Universal Robots PolyScope program: nastrobello.urp

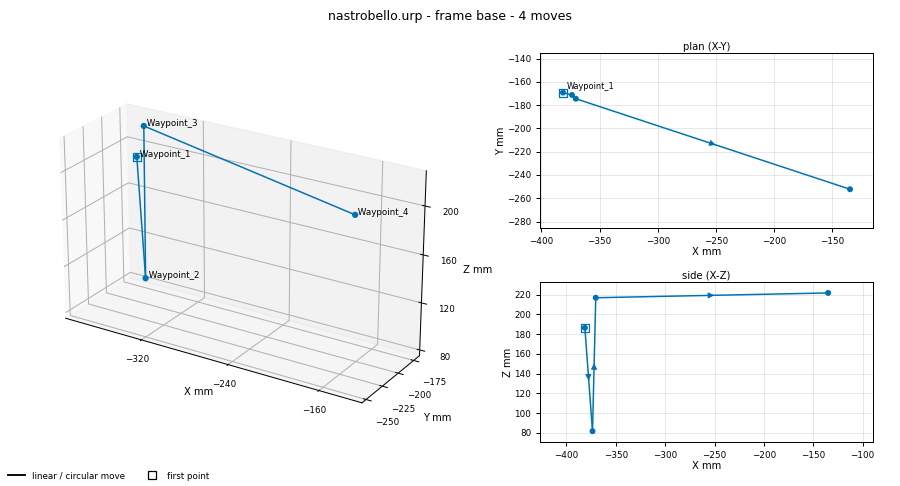
[picture p0: tool path of nastrobello.urp in frame base, 4 of 4 moves have a stored position in this frame; points joined in program order, loops and branches not executed]
Program nastrobello (installation=default directory=/programs createdIn=3.15.8.106339 lastSavedIn=3.15.8.106339 robotSerialNumber=2021330429)
Calibrated DH parameters: a=[-0.000156, -0.236402, -0.171625, 0.000006, -0.000047, 0]; d=[0.151683, 29.702709, 78.973085, -108.563557, 0.085229, 0.082167]; alpha=[1.57015, 0.001987, 0.001164, 1.571718, -1.571778, 0]; deltaTheta=[-0.000066, 0.24449, 0.39032, -0.635025, 0.000068, -0.000043]
Robot Program (runOnlyOnce=false)
  URCap Gripper Activate (Robotiq_Grippers, Robotiq Inc.) dataModel(ResetAndActivateKey=false)
  URCap Gripper (Robotiq_Grippers, Robotiq Inc.) dataModel(position=0.0, force=0.0, speed=0.0, positionInDouble=0.0, forceInDouble=0.0, speedInDouble=0.0, slaveIds=[9], blocking=true)
  Timer (action=Stop) variable(name=volo)
  ready := False
  engineon := digital_out[0]
  engineon := False
  sensoreBasso := digital_in[4]
  sensoreAlto := digital_in[6]
  sensoreStop := digital_in[5]
  tempoVolo := 4000
  Loop Forever
    If digital_in[4]== True
      engineon := True
      Wait DigitalInput pin=digital_in[4]; digitalValue=0
    ElseIf digital_in[6]== True
      engineon := True
      Wait DigitalInput pin=digital_in[6]; digitalValue=0
    ElseIf digital_in[5]== True
      engineon := False
      MoveL speed 250 mm/s, acceleration 1200 mm/s^2 (useActiveTCP=true) feature=Base
        Waypoint Waypoint_1: TCP in base x=-381.388 y=-169.307 z=186.364 mm, rx=0.0312 ry=3.0921 rz=-0.0497 rad; joints [217.72, -119.894, -42.767, -108.34, 93.283, 308.738] deg; flange x=-389.019 y=-164.19 z=343.095 mm, rx=0.0312 ry=3.0921 rz=-0.0497 rad
      MoveL speed 250 mm/s, acceleration 1200 mm/s^2 (useActiveTCP=true) feature=Base
        Waypoint Waypoint_2: TCP in base x=-373.641 y=-171.323 z=81.625 mm, rx=0.0313 ry=3.0921 rz=-0.0497 rad; joints [218.633, -116.939, -75.878, -78.131, 93.316, 309.678] deg; flange x=-381.271 y=-166.208 z=238.356 mm, rx=0.0313 ry=3.0921 rz=-0.0497 rad
      URCap Gripper (Robotiq_Grippers, Robotiq Inc.) dataModel(position=51.372549019607845, force=0.0, speed=0.0, positionInDouble=51.372549019607845, forceInDouble=0.0, speedInDouble=0.0, slaveIds=[9], blocking=true)
      MoveL speed 250 mm/s, acceleration 1200 mm/s^2 (useActiveTCP=true) feature=Base
        Waypoint Waypoint_3: TCP in base x=-370.357 y=-174.548 z=216.862 mm, rx=0.032 ry=3.0975 rz=-0.044 rad; joints [219.476, -120.992, -32.181, -117.632, 92.948, 310.521] deg; flange x=-377.159 y=-170.022 z=373.65 mm, rx=0.032 ry=3.0975 rz=-0.044 rad
      MoveL speed 250 mm/s, acceleration 1200 mm/s^2 (useActiveTCP=true) feature=Base
        Waypoint Waypoint_4: TCP in base x=-134.875 y=-252.278 z=221.727 mm, rx=0.0321 ry=3.0975 rz=-0.0439 rad; joints [262.666, -83.874, -78.503, -106.241, 92.71, 353.777] deg; flange x=-141.677 y=-247.765 z=378.514 mm, rx=0.0321 ry=3.0975 rz=-0.0439 rad
      Pallet pattern(dimensionality=Square firstAxisCount=2 secondAxisCount=2 thirdAxisCount=5 motionType=MoveL speed=0.25 acceleration=1.2 useActiveTCP=true, counterVariable(name=cnt_1, initializeExpression=0), patternPoseVariable(name=pose_1), feature=Base, children(Waypoint(type=Fixed name=Corner1_1, position(joints=4.717325687408447, -2.232218090687887, -1.3913286367999476, -1.0653889814959925, 1.6609495878219604, 6.306212246661083 pose=-0.08976236359262711, -0.4291511389600013, 0.009188706301395622, 0.027577147014370685, 3.053416589492967, -0.0321823131281283), poseInFeatureCoordinates=[-0.089762, -0.429151, 0.009189, 0.027577, 3.053417, -0.032182], outputFlangePose=[-0.103511, -0.425724, 0.165548, 0.027577, 3.053417, -0.032182]), Waypoint(type=Fixed name=Corner2_1, position(joints=5.005774021148682, -2.179821316395895, -1.48505145708193, -0.9999783674823206, 1.6508749723434448, 6.595563862715856 pose=0.03118660998664156, -0.4291712110429884, 0.011085502208470405, 0.02761157513313603, 3.053453182136718, -0.032263865589663966), poseInFeatureCoordinates=[0.031187, -0.429171, 0.011086, 0.027612, 3.053453, -0.032264], outputFlangePose=[0.017444, -0.425736, 0.167445, 0.027612, 3.053453, -0.032264]), Waypoint(type=Fixed name=Corner3_1, position(joints=5.060262680053711, -1.948681656514303, -1.8695586363421839, -0.8424580732928675, 1.647793173789978, 6.650210444127218 pose=0.031156149701591744, -0.36408695526798923, 0.01105682758960308, 0.027631286382420437, 3.0534637137929583, -0.03225085570525061), poseInFeatureCoordinates=[0.031156, -0.364087, 0.011057, 0.027631, 3.053464, -0.032251], outputFlangePose=[0.017415, -0.360653, 0.167417, 0.027631, 3.053464, -0.032251]), Waypoint(type=Fixed name=Corner4_1, position(joints=4.718104839324951, -2.0136664549456995, -1.7641990820514124, -0.9110310713397425, 1.6604578495025635, 6.3069676275001925 pose=-0.08976155355196079, -0.3665535168441274, 0.009168617974270987, 0.027481938486564293, 3.053493094310215, -0.032138841944468574), poseInFeatureCoordinates=[-0.089762, -0.366554, 0.009169, 0.027482, 3.053493, -0.032139], outputFlangePose=[-0.103499, -0.363132, 0.165529, 0.027482, 3.053493, -0.032139]))); actionSequence(name=PalletSequence motionType=MoveL speed=0.25 acceleration=1.2 useActiveTCP=true, anchorWaypoint(type=Fixed name=PatternPoint_1, position(joints=4.718020915985107, -1.8602607885943812, -1.0282829443561, -1.8004000822650355, 1.659809947013855, 6.3059250007020395 pose=-0.08975527979420515, -0.36654202546761244, 0.20249238196803704, 0.027482330613282577, 3.0534311557917384, -0.03220644890340183), poseInFeatureCoordinates=[-0.089755, -0.366542, 0.202492, 0.027482, 3.053431, -0.032206], outputFlangePose=[-0.103502, -0.363113, 0.358852, 0.027482, 3.053431, -0.032206]), feature=Base, children(Waypoint(type=Fixed name=Approach_1, position(joints=4.717973232269287, -1.860248867665426, -1.0282467047320765, -1.8003881613360804, 1.6597744226455688, 6.30596095347871 pose=-0.08978118139786681, -0.3665466262118018, 0.20250783773884545, 0.027606886294300952, 3.053463920443164, -0.032300040654198), poseInFeatureCoordinates=[-0.089781, -0.366547, 0.202508, 0.027607, 3.053464, -0.0323], outputFlangePose=[-0.103522, -0.363108, 0.358868, 0.027607, 3.053464, -0.0323]), Waypoint=PatternPoint_1, Set(type=NoAction), Wait(type=Condition, expression=volo>tempoVolo), Waypoint(type=Fixed name=Exit_1, position(joints=4.718020915985107, -1.8602607885943812, -1.0282586256610315, -1.8004120031939905, 1.6597744226455688, 6.30593698496093 pose=-0.08976373110781001, -0.3665437027494239, 0.2024977765553612, 0.027500770851460146, 3.053466015947447, -0.032225658991452605), poseInFeatureCoordinates=[-0.089764, -0.366544, 0.202498, 0.027501, 3.053466, -0.032226], outputFlangePose=[-0.103505, -0.363113, 0.358858, 0.027501, 3.053466, -0.032226])))
        Pattern -> pattern
        AnchoredSequence -> PalletSequence
      Timer (action=Start) variable=volo
      Timer (action=Reset) variable=volo
    ElseIf volo>tempoVolo
      Timer (action=Stop) variable=volo
      Timer (action=Reset) variable=volo
